Staubli VAL3: get.pgx

public program get(string& x_sItem[], num x_nIndex)
  local string l_sKey
  local num i
  local string l_sItem
begin
  // start from the first
  l_sKey=first(pt:tTraj)
  // search it
  while l_sKey!=""
    x_sItem=l_sKey
    l_sKey=next(pt:tTraj[l_sKey])
    if i==x_nIndex
      return
    else
      i=i+1
    endIf
  endWhile
end
